FUNCTION_BLOCK OpeningValveDurLogic (* CAT Function Block Type *)
  (* Standard: 61499-2 *)
  (* Version 0.0, 6/26/2026, Schneider Electric, template *)
  PACKAGE SE.Nereda;
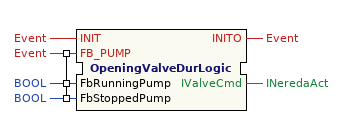
  EVENT_INPUT
    INIT;
    FB_PUMP WITH FbRunningPump, FbStoppedPump; (* Normal Execution Request *)
  END_EVENT
  EVENT_OUTPUT
    INITO;
  END_EVENT
  VAR_INPUT
    FbRunningPump : BOOL;
    FbStoppedPump : BOOL;
  END_VAR
  PLUGS
    IValveCmd : INeredaAct;
  END_PLUGS
  (* 01 - FUNCTIONNAL INPUT INTERFACE *)
  (* 00 - INITIALIZATION *)
  (* 05 - LOGIC *)
  (* 06 - HMI INTERFACE *)
  (* 03 - FIELD INTERFACE *)
  (* 02 - FUNCTIONNAL OUTPUT INTERFACE *)
  (* Calamity Valve Logic *)
  FBS
    ValveLogic : OpeningValveBasic;
    ValveCmd : boolValueChanged;
    OpeningValveDur : E_DELAY_V_D;
    IThis : OpeningValveDurLogic_HMI(QI := TRUE);
    RESET_BTNs : RESET_BTNs;
    Valve : BOOL2INT;
  END_FBS
  EVENT_CONNECTIONS
    INIT TO IThis.45DF0F05DD2E6916;
    OpeningValveDur.INITO TO INITO;
    ValveLogic.08F74931246E5910 TO IThis.E845F16C24CB67B1;
    RESET_BTNs.920962203CA54948 TO IThis.3C12A0D93D14CDE4;
    OpeningValveDur.INITO TO IThis.8639AE2A08C86ED3;
    IThis.9ADA932D5BFA8E47 TO OpeningValveDur.INIT;
    IThis.16D83178296B5D7E TO ValveLogic.D549B502E1232CDF;
    IThis.16D83178296B5D7E TO RESET_BTNs.AB695E9A35A20E19;
    FB_PUMP TO ValveLogic.AA2535F1FE364DBC;
    IValveCmd.9CD053F8408797ED TO ValveLogic.71DE2BDA4EE82470;
    IValveCmd.CC753684FA882790 TO ValveLogic.71DE2BDA4EE82470;
    OpeningValveDur.1457E63E0C241C83 TO ValveLogic.56FEED5D7757F0A3;
    ValveLogic.E7B2313E02E11A39 TO ValveCmd.REQ;
    ValveCmd.CHD TO Valve.DD5870AA881150BB;
    ValveLogic.01695A2546E5DEDD TO OpeningValveDur.START;
    ValveLogic.5860258CFE1E31BC TO OpeningValveDur.STOP;
    Valve.6FC99A5BD1C38561 TO IValveCmd.0F1CDF9A9B4A227A;
    IThis.3DD19A06F40F70E1 TO OpeningValveDur.8C325F07198FCB13;
  END_CONNECTIONS
  DATA_CONNECTIONS
    ValveLogic.4AC0A9927738781F TO IThis.990A6D7C96184C76;
    IThis.A53C89DB96DE7793 TO OpeningValveDur.DT1;
    IThis.8902C21ADB31D3BD TO ValveLogic.CFC90A7FF1CE9B71;
    IThis.8902C21ADB31D3BD TO RESET_BTNs.479D4538AEFD6EE1;
    FbRunningPump TO ValveLogic.6F3653F02BAF1FDA;
    FbStoppedPump TO ValveLogic.2B74E1411E640D68;
    IValveCmd.7F6CC7FEB9223DF3 TO ValveLogic.2A5667F4487C2CF2;
    IValveCmd.A8D6C4A1FDCCA991 TO ValveLogic.1ECB3193CD72FEBA;
    IValveCmd.8A8A07EFCDA1443C TO ValveLogic.AA00379C07DC4373;
    OpeningValveDur.716D3F3042596C89 TO ValveLogic.7B2E2342833916F8;
    ValveLogic.C4B3168A8E5A064C TO ValveCmd.Input;
    ValveCmd.Output TO Valve.4573FC8F228EB71D;
    Valve.A6DEF5F9C27C1848 TO IValveCmd.710D7FC54EE3F35A;
  END_CONNECTIONS
END_FUNCTION_BLOCK
